INTERFACE I_IgnoreInitRegistration EXTENDS __System.IQueryInterface

END_INTERFACE

(* stored: Version 1.1.0.1
   Itf I_IgnoreInitRegistration: Id {55cd1db4-db2b-4ea8-a2a7-0dee57f9c87b} *)
